Fanuc TP program (LS listing): PRSHIFT.LS

/PROG  PRSHIFT
/ATTR
OWNER		= MNEDITOR;
COMMENT		= "PrShift";
PROG_SIZE	= 0;
CREATE		= DATE 26-01-01  TIME 00:00:00;
MODIFIED	= DATE 26-01-01  TIME 00:00:00;
FILE_NAME	= ;
VERSION		= 0;
LINE_COUNT	= 6;
MEMORY_SIZE	= 0;
PROTECT		= READ_WRITE;
TCD:  STACK_SIZE	= 0,
      TASK_PRIORITY	= 50,
      TIME_SLICE	= 0,
      BUSY_LAMP_OFF	= 0,
      ABORT_REQUEST	= 0,
      PAUSE_REQUEST	= 0;
DEFAULT_GROUP	= 1,*,*,*,*;
CONTROL_CODE	= 00000000 00000000;
/MN
   1:  !RAPID PointRefProbe.PrShift ;
   2:  PR[99,2]=PR[99,2]+50    ;
   3:  UFRAME_NUM=0 ;
   4:  UTOOL_NUM=1 ;
   5:L PR[99] 400mm/sec FINE    ;
   6:  R[1:prSteps]=R[1:prSteps]+1    ;
/POS
/END
